# EPICS substitutions: siteApps-725b29e158e8061764313f5708af9e46fe30c0a8/siteApps-725b29e158e8061764313f5708af9e46fe30c0a8/Tr6/tr6App/Db/user.substitutions
# Example substitutions file

file "db/dbExample1.db" {
    { user = "silee" }
}

file db/dbExample2.db {
    pattern { user, no, scan }
        { "silee", 1, "1 second" }
        { "silee", 2, "2 second" }
        { "silee", 3, "5 second" }
}
